FUNCTION_BLOCK L3_L2CommPlug (* Composite Function Block Type *)
  (* Standard: 61499-2 *)
  (* Version 0.0, 2014-11-25, EQUEROL, UJI *)
  (* Version 1.0, 2015-01-08, EQUEROL, UJI, modified adapter definition *)
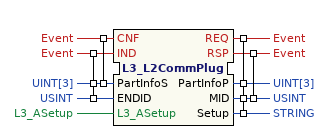
  EVENT_INPUT
    CNF WITH PartInfoS; (* Initialization Request *)
    IND WITH PartInfoS, ENDID; (* Normal Execution Request *)
  END_EVENT
  EVENT_OUTPUT
    REQ WITH PartInfoP, MID, Setup; (* Initialization Confirm *)
    RSP WITH MID; (* Execution Confirmation *)
  END_EVENT
  VAR_INPUT
    PartInfoS : ARRAY [0..2] OF UINT; (* Part ID, family, type *)
    ENDID : USINT; (* Setup execution returned code *)
  END_VAR
  VAR_OUTPUT
    PartInfoP : ARRAY [0..2] OF UINT; (* Part ID, Family, Type *)
    MID : USINT; (* Destination machine identifier *)
    Setup : STRING; (* Subphase to be trasmitted *)
  END_VAR
  SOCKETS
    L3_ASetup : L3_ASetup;
  END_SOCKETS
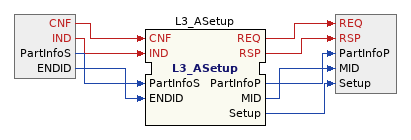
  EVENT_CONNECTIONS
    CNF TO L3_ASetup.CNF;
    IND TO L3_ASetup.IND;
    L3_ASetup.REQ TO REQ;
    L3_ASetup.RSP TO RSP;
  END_CONNECTIONS
  DATA_CONNECTIONS
    PartInfoS TO L3_ASetup.PartInfoS;
    ENDID TO L3_ASetup.ENDID;
    L3_ASetup.PartInfoP TO PartInfoP;
    L3_ASetup.MID TO MID;
    L3_ASetup.Setup TO Setup;
  END_CONNECTIONS
END_FUNCTION_BLOCK
